# EPICS StreamDevice protocol: RSpowerm/device_config/RSpowerm.proto
Terminator = CR LF;

ReplyTimeout = 2000;

@init { out "SYST:PRES"; wait 2000; }

getDevIdent {
   out "*IDN?";
   in "%40c";
}

getFreq {
   out "SENSE\$1:FREQ?";
   in "%f";
}

setFreq {
   out "SENSE\$1:FREQ %f";
   @init { out "SENSE\$1:FREQ 1.3 GHz"; getFreq; }
}

getPower {
#   out "DISP:WIND:SEL \$1";
   out "MEAS\$1:SCAL:POW:AVG? (@\$1)";
   in "%f";
}

setDisp {
   out "DISP:ILL %{0|1}";
   @init { out "DISP:ILL 1"; out "DISP:WIND2: ON";}
}

getStatQuesCond {
   out "STAT:QUES:COND?";
   in "%d";
}

#frequently changing potocol files can be reloaded; without record argument all records
#epics> streamReload()

#http://epics.web.psi.ch/software/streamdevice/doc/protocol.html
